Staubli VAL3: start.pgx

program start()
begin
  // feedback task will run every 32 ms (approx. 31 Hz)
  nFbkPeriod=0.032
  //nFbkPeriod = 0.05
  //nFbkPeriod = 1.0

  // motion task will run every 12 ms (approx. 83 Hz)
  //nMotionPeriod=0.012
  //nMotionPeriod = 0.05
  nMotionPeriod = 0.004

  nTrajReception = 0.004
  // not in use at the moment
  nScreenUpdate = 1.0

  nDeg2Rad = 3.14159265359 / 180.0
  nRad2Deg = 180.0 / 3.14159265359

  sStreamTaskName = "streamerTask"
  sTrajPtTaskName = "trajPtTask"
  sMotionTaskName = "motionTask"
  sScreenTaskName = "screenTask"
  sHtbtTaskName = "htbtTask"

  // initialise TCP/IP parameters
  call initParams()
  // setup prefix and header of ROS messages
  call setupRosMsgs()

  // socket connections: initially disconnected
  nDataIn = 0
  nDataOut = 0

  // flags to control tasks: should start sending/receiving
  bSendData = true
  bRecvData = true
  bCheckHeartbeat = false

  nPtsPopped = 0
  nMovePts = 0

  // debug status
  nDebugStatus = 0

  // ensure motion buffer is empty
  call libTrajPtBuffer:clear()
  call libMoveBuffer:clear()

  // before anything else, enable power (only works if robot is in remote mode)
  //enablePower()
  //if (watch(isPowered(), 5) == false)
  //  popUpMsg("Arm power could not be enabled")
  //endIf

  // create joint state and robot status streamer task to send data to industrial_robot_client
  taskCreateSync sStreamTaskName, nFbkPeriod, bFbkOverrun, dataStreamer()

  // create trajectory point task to receive data from industrial_robot_client
  taskCreateSync sTrajPtTaskName, nTrajReception, bTrajPtOverrun, dataReceiver()

  // create motion task to synchronously apply motion commands to robot
  taskCreateSync sMotionTaskName, nMotionPeriod, bMotionOverrun, motionControl()

  // create synchronous task to update screen
  //taskCreateSync sScreenTaskName, nScreenUpdate, bScreenOverrun, screenUpdate()
  taskCreate sScreenTaskName, 10, screenUpdate()

  // create asynchronous task to receive heartbeat on port 11002
  taskCreate sHtbtTaskName, 10, recvHeartbeat()

end
